// TIA Portal V16 export
// export: Created 2021-09-07T10:36:59.5125101Z, ExportSetting WithDefaults, DisplayName Totally Integrated Automation Portal, DisplayVersion V16 Update 3, DisplayName TIA Portal Version Control Interface, DisplayVersion V16 Update 2, DisplayName TIA Portal Openness, DisplayVersion V16 Update 3, DisplayName TIA Portal Teamcenter Gateway, DisplayVersion V16, DisplayName STEP 7 Professional, DisplayVersion V16 Update 3, DisplayName STEP 7 Safety, DisplayVersion V16, DisplayName WinCC Advanced, DisplayVersion V16 Update 3
DATA_BLOCK "AllFlowCounter_DB"   // DB23
VERSION : 0.1
// stored: AutoNumber true, DBAccessibleFromOPCUA true, InstanceOfName AllFlowCounter, InstanceOfType FB
"AllFlowCounter"
   // VAR
   //    prewHour : USInt;
   //    prewDay : USInt;
   //    FM201 { S7_SetPoint := 'True'} : "VolumeCounter";
   //    FM501 { S7_SetPoint := 'True'} : "VolumeCounter";
   //    FM502 { S7_SetPoint := 'True'} : "VolumeCounter";
   //    FM901 { S7_SetPoint := 'True'} : "VolumeCounter";
   //    FM902 { S7_SetPoint := 'True'} : "VolumeCounter";
   //    FM1201 { S7_SetPoint := 'True'} : "VolumeCounter";
   //    FM1301 { S7_SetPoint := 'True'} : "VolumeCounter";
   //    FM1302 { S7_SetPoint := 'True'} : "VolumeCounter";
   //    FM1701 { S7_SetPoint := 'True'} : "VolumeCounter";
   //    FM1801 { S7_SetPoint := 'True'} : "VolumeCounter";
   // END_VAR
BEGIN
END_DATA_BLOCK
